// TIA Portal V20 export
DATA_BLOCK "SP202"   // DB345
// stored: MemoryReserve 100
   VAR
      "AUTO INITIATE PBL LAMP (GREEN)" : Bool := FALSE;
      "STOP PBL LAMP ON (RED)" : Bool := TRUE;
      SPARE_4 : Bool := FALSE;
      "ENABLE PBL LAMP ON (WHITE)" : Bool := FALSE;
      "SAFETY RESET PBL LAMP (BLUE)" : Bool := FALSE;
      SPARE : Bool := FALSE;
      SPARE_1 : Bool := FALSE;
      SPARE_2 : Bool := FALSE;
      "TOWER LAMP 1 ON (RED)" : Bool := TRUE;
      "TOWER LAMP 2 ON (AMBER)" : Bool := FALSE;
      "TOWER LAMP 3 ON (GREEN)" : Bool := FALSE;
      "TOWER LAMP 4 ON (WHITE)" : Bool := FALSE;
      "TOWER LAMP 5 ON (BLUE)" : Bool := FALSE;
      "Buzzer On" : Bool := FALSE;
      SPARE_3 : Bool := FALSE;
      SPARE_5 : Bool := FALSE;
   END_VAR
BEGIN
END_DATA_BLOCK
